Yaskawa INFORM job: ARLO.JBI

/JOB
//NAME ARLO
//POS
///NPOS 91,0,0,0
///TOOL 0
///PULSE
C000=8847,58516,-58779,12036,431,10843
C001=8069,58299,-59170,12245,373,10789
C002=7517,58014,-59957,12397,227,10697
C003=7822,57735,-61005,12323,18,10585
C004=9866,57622,-61273,11789,-33,10553
C005=10429,57501,-62373,11637,-221,10414
C006=10690,56513,-62168,11570,-185,10435
C007=11215,56943,-62715,11427,-268,10360
C008=11014,56967,-62376,11484,-214,10405
C009=10663,57036,-62627,11574,-261,10376
C010=10834,57045,-62928,11526,-309,10336
C011=10690,54801,-61796,11572,-122,10482
C012=11166,57065,-62703,11442,-266,10363
C013=11166,56428,-62591,11443,-248,10378
C014=8957,55552,-61363,12028,-51,10540
C015=7955,57255,-61765,12289,-129,10498
C016=8251,57221,-61472,12213,-71,10530
C017=8662,57236,-61524,12105,-81,10524
C018=9003,57191,-61964,12014,-160,10471
C019=8611,57018,-62701,12110,-302,10388
C020=8715,56966,-63449,12072,-441,10300
C021=9299,56966,-63438,11920,-427,10293
C022=9671,56977,-63233,11826,-382,10313
C023=10045,57107,-62765,11734,-293,10367
C024=10045,56434,-62648,11735,-272,10382
C025=8454,56167,-62546,12153,-276,10407
C026=7474,57171,-61784,12416,-137,10498
C027=8065,57012,-63291,12247,-426,10327
C028=8112,56995,-63710,12227,-505,10278
C029=7536,56991,-63959,12373,-567,10260
C030=7062,56998,-63609,12504,-508,10306
C031=6479,57154,-61893,12675,-164,10490
C032=6479,56360,-61754,12676,-135,10504
C033=6090,57110,-62033,12777,-196,10478
C034=5719,57093,-62160,12873,-226,10468
C035=5429,57029,-62733,12944,-352,10416
C036=5752,56968,-63873,12843,-591,10302
C037=6393,56967,-64213,12668,-648,10255
C038=7156,56967,-63934,12473,-573,10270
C039=6957,56966,-64011,12524,-593,10266
C040=5977,57107,-62055,12806,-202,10477
C041=5977,56557,-61960,12807,-182,10486
C042=5217,56417,-63430,12991,-506,10354
C043=5217,56953,-63525,12990,-526,10345
C044=5037,56996,-62827,13046,-377,10412
C045=4759,57064,-62197,13123,-241,10473
C046=4147,57045,-62351,13282,-280,10464
C047=3912,56991,-62885,13339,-403,10421
C048=4171,56942,-64156,13253,-685,10309
C049=4768,56945,-64414,13091,-729,10272
C050=5336,56942,-64263,12945,-683,10273
C051=5497,56942,-63945,12909,-611,10300
C052=5200,56998,-63094,12999,-434,10386
C053=5115,55703,-62996,13023,-412,10396
C054=4019,56474,-64224,13293,-704,10306
C055=4034,56920,-64373,13287,-737,10293
C056=3684,56936,-62563,13404,-332,10449
C057=3194,56973,-62664,13532,-361,10446
C058=2889,56939,-63075,13608,-460,10418
C059=2924,56924,-63322,13595,-518,10399
C060=3841,56917,-63464,13353,-538,10373
C061=3137,56906,-64361,13523,-755,10314
C062=3137,56485,-64287,13524,-738,10320
C063=2620,56906,-63456,13673,-554,10393
C064=2687,56893,-63954,13649,-670,10355
C065=2242,56895,-64283,13761,-755,10341
C066=1731,56896,-63838,13902,-657,10383
C067=1657,56938,-62956,13931,-446,10443
C068=1244,56974,-62561,14042,-354,10474
C069=790,56930,-63067,14157,-481,10449
C070=824,56895,-63926,14139,-690,10397
C071=1335,56897,-64394,13997,-797,10356
C072=1716,56898,-63767,13906,-640,10388
C073=1713,56564,-63682,13908,-621,10395
C074=1650,56605,-62925,13932,-440,10446
C075=1650,56971,-62989,13932,-455,10442
C076=2056,57020,-62465,13830,-326,10473
C077=2565,56979,-62893,13693,-423,10437
C078=2656,56939,-63593,13662,-586,10384
C079=2656,56617,-63537,13663,-573,10388
C080=792,56525,-64349,14142,-795,10374
C081=792,56934,-64421,14141,-813,10370
C082=456,57013,-62533,14249,-354,10486
C083=-135,56960,-63152,14400,-511,10460
C084=-821,57027,-62404,14585,-328,10505
C085=-906,56933,-64388,14591,-828,10415
C086=-906,55857,-64186,14593,-777,10424
C087=-1179,55863,-64487,14661,-857,10418
C088=-1179,56858,-64676,14659,-904,10410
C089=4084,56971,-64449,13272,-758,10285
C090=4084,56223,-64314,13275,-728,10297
//INST
///DATE 2014/09/21 00:35
///ATTR 0,0,0,0,0,0,0,0,0,0,0,0,0,1,0,0
///FRAME BASE
NOP
JUMP *S
MOVJ C000 VJ=25.00 PL=0
MOVJ C001 VJ=25.00 PL=0
MOVJ C002 VJ=25.00 PL=0
MOVJ C003 VJ=25.00 PL=0
MOVJ C004 VJ=25.00 PL=0
MOVJ C005 VJ=25.00 PL=0
MOVJ C006 VJ=50.00 CONT
MOVJ C007 VJ=25.00 CONT
MOVJ C008 VJ=25.00 CONT
MOVJ C009 VJ=25.00 CONT
MOVJ C010 VJ=25.00 CONT
MOVJ C011 VJ=50.00 CONT
MOVJ C012 VJ=50.00 CONT
MOVJ C013 VJ=50.00 CONT
*S
MOVJ C014 VJ=50.00 CONT
PAUSE
MOVJ C015 VJ=10.00 CONT
MOVJ C016 VJ=10.00 CONT
MOVJ C017 VJ=10.00 CONT
MOVJ C018 VJ=10.00 CONT
MOVJ C019 VJ=10.00 CONT
MOVJ C020 VJ=10.00 CONT
MOVJ C021 VJ=10.00 CONT
MOVJ C022 VJ=10.00 CONT
MOVJ C023 VJ=10.00 CONT
MOVJ C024 VJ=10.00 CONT
MOVJ C025 VJ=10.00 CONT
MOVJ C026 VJ=10.00 PL=4
MOVJ C027 VJ=10.00 CONT
MOVJ C028 VJ=10.00 CONT
MOVJ C029 VJ=10.00 CONT
MOVJ C030 VJ=10.00 CONT
MOVJ C031 VJ=10.00 CONT
MOVJ C032 VJ=10.00 CONT
MOVJ C033 VJ=10.00 CONT
MOVJ C034 VJ=10.00 CONT
MOVJ C035 VJ=10.00 CONT
MOVJ C036 VJ=10.00 CONT
MOVJ C037 VJ=10.00 CONT
MOVJ C038 VJ=10.00 CONT
MOVJ C039 VJ=10.00 CONT
MOVJ C040 VJ=10.00 CONT
MOVJ C041 VJ=10.00 CONT
MOVJ C042 VJ=10.00 CONT
MOVJ C043 VJ=10.00 CONT
MOVJ C044 VJ=10.00 CONT
MOVJ C045 VJ=10.00 CONT
MOVJ C046 VJ=10.00 CONT
MOVJ C047 VJ=10.00 CONT
MOVJ C048 VJ=10.00 CONT
MOVJ C049 VJ=10.00 CONT
MOVJ C050 VJ=10.00 CONT
MOVJ C051 VJ=10.00 CONT
MOVJ C052 VJ=10.00 PL=4
MOVJ C053 VJ=10.00 CONT
MOVJ C054 VJ=10.00 CONT
*R
MOVJ C055 VJ=5.00 CONT
MOVJ C056 VJ=5.00 CONT
MOVJ C057 VJ=10.00 CONT
MOVJ C058 VJ=10.00 CONT
MOVJ C059 VJ=10.00 CONT
MOVJ C060 VJ=10.00 CONT
MOVJ C061 VJ=10.00 CONT
MOVJ C062 VJ=10.00 CONT
*OO
MOVJ C063 VJ=10.00 CONT
MOVJ C064 VJ=10.00 CONT
MOVJ C065 VJ=10.00 CONT
MOVJ C066 VJ=10.00 CONT
MOVJ C067 VJ=10.00 CONT
MOVJ C068 VJ=10.00 CONT
MOVJ C069 VJ=10.00 CONT
MOVJ C070 VJ=10.00 CONT
MOVJ C071 VJ=5.00 CONT
MOVJ C072 VJ=5.00 CONT
MOVJ C073 VJ=10.00 CONT
MOVJ C074 VJ=10.00 CONT
MOVJ C075 VJ=10.00 CONT
MOVJ C076 VJ=10.00 CONT
MOVJ C077 VJ=10.00 CONT
MOVJ C078 VJ=10.00 CONT
MOVJ C079 VJ=10.00 CONT
MOVJ C080 VJ=10.00 CONT
MOVJ C081 VJ=10.00 CONT
MOVJ C082 VJ=10.00 CONT
MOVJ C083 VJ=10.00 CONT
MOVJ C084 VJ=10.00 CONT
MOVJ C085 VJ=10.00 CONT
MOVJ C086 VJ=10.00 CONT
MOVJ C087 VJ=25.00 CONT
MOVJ C088 VJ=25.00 CONT
MOVJ C089 VJ=25.00 CONT
MOVJ C090 VJ=25.00 CONT
JUMP *S
END
